PROGRAM FUN_DisconnectVPN

VAR_INPUT
	ParamNetID				: STRING :='' ; // Unit ID of the PC with internet connexion
	IN_CmdStart 			: BOOL;
	IN_DirExe				: STRING;
END_VAR
VAR_OUTPUT
	OUT_Completed			: BOOL;
END_VAR

VAR
	TRIG_Start				: R_TRIG;
	start_process			: NT_StartProcess;
END_VAR

TRIG_Start(ClK := IN_CmdStart);

start_process
(
	NETID := ParamNetID,
	PATHSTR := '"c:\Program Files\OpenVPN\bin\openvpn-gui.exe" ',
	DIRNAME := 'C:\Program Files\OpenVPN\bin',
	COMNDLINE := '--command disconnect_all',
	Start := TRIG_Start.Q
);

END_PROGRAM

(* stored: Version 1.1.0.1, ProductVersion 3.1.4024.6
   POU FUN_DisconnectVPN: Id {c8ed6f7b-d817-4306-af09-c9af7b878675}, SpecialFunc None *)
